(* Logix 5000 project; controller LIgacoesEletricas vendor 1 type 14 code 43 rev 13.1; software revision 13.00 *)

TASK MainTask (continuous, watchdog 500 ms) : MainProgram

MODULES
   Controller : vendor 1 type 14 code 43 (CompactLogixController 0, rev 13.1)
      Local : CompactBus (CompactVirtualAdapter 3, rev 13.1, Input RPI 2 ms)
         M1 : 1769-IQ16 (Compact 1, rev 1.1, Input RPI 2 ms)   // Módulo 1
         M3 : 1769-IQ16 (Compact 3, rev 1.1, Input RPI 2 ms)   // Módulo 3
         M2 : 1769-IQ16 (Compact 2, rev 1.1, Input RPI 2 ms)   // Módulo 2
         M4 : vendor 1 type 7 code 86 (Compact 4, rev 2.1, Output RPI 2 ms)   // Módulo 4
         M5 : vendor 1 type 7 code 86 (Compact 5, rev 2.1, Output RPI 2 ms)   // Módulo 5
         M7 : vendor 1 type 7 code 86 (Compact 7, rev 2.1, Output RPI 2 ms)   // Módulo 7
         M6 : vendor 1 type 7 code 86 (Compact 6, rev 2.1, Output RPI 2 ms)   // Módulo 6
END_MODULES

VAR_GLOBAL   (* controller tags *)
   E0 : ALIAS FOR Local:1:I.Data.0;   // E0 - Entrada do painel
   E1 : ALIAS FOR Local:1:I.Data.1;   // E1 - Entrada do painel
   E1B1 : ALIAS FOR Local:1:I.Data.8;   // E1B1 - indicação de cilindro S1Y1 recuado - alimentação de peças
   E1B2 : ALIAS FOR Local:1:I.Data.9;   // E1B2 - Iindicação do cilindro S1Y1 avançado - alimentação de peças
   E1S1 : ALIAS FOR Local:1:I.Data.10;   // E1S1 - indicação de presença de peças na alimentação
   E1S2 : ALIAS FOR Local:1:I.Data.11;   // E1S2 - indicação de presença de peças fixada na ventosa - oscilador
   E1S3 : ALIAS FOR Local:1:I.Data.12;   // E1S3 - indicação do oscilador (S1Y5) no lado do alimentador
   E1S4 : ALIAS FOR Local:1:I.Data.13;   // E1S4 - indicação do oscilador (S1Y4) no lado do elevador
   E2 : ALIAS FOR Local:1:I.Data.2;   // E2 - Entrada do painel
   E2B1 : ALIAS FOR Local:1:I.Data.14;   // E2B1 - indicação da plataforma (S2Y1) no nível inferior
   E2B2 : ALIAS FOR Local:1:I.Data.15;   // E2B2 - indicação da plataforma (S2Y2) no nível superior
   E2B3 : ALIAS FOR Local:2:I.Data.4;   // E2B3 - indicação do cilindro S2Y3 recuado - descarga de peças na seleção
   E2B4 : ALIAS FOR Local:2:I.Data.5;   // E2B4 - indicação do cilindro S2Y3 avançado - descarga de peças na seleção
   E2B5 : ALIAS FOR Local:2:I.Data.6;   // E2B5 - indicação de peças da cor laranja - sensor ótico - seleção
   E2B6 : ALIAS FOR Local:2:I.Data.7;   // E2B6 - indicação de presença de peças - sensor capacitivo - seleção
   E2B7 : ALIAS FOR Local:2:I.Data.8;   // E2B7 - indicação de peças metálicas - sensor indutivo - seleção
   E3 : ALIAS FOR Local:1:I.Data.3;   // E3 - Entrada do painel
   E3B1 : ALIAS FOR Local:2:I.Data.9;   // E3B1 - indicação de furadeira (S3Y1) na posição superior
   E3B2 : ALIAS FOR Local:2:I.Data.10;   // E3B2 - Iindicação da furadeira (S3Y2) na posição inferior
   E3B3 : ALIAS FOR Local:2:I.Data.0;   // E3B3 - indicação do cilindro S3Y3 recuado - controle de qualidade
   E3B4 : ALIAS FOR Local:2:I.Data.1;   // E3B4 - indicação do cilindro S3Y3 avançado - controle de qualidade
   E3B5 : ALIAS FOR Local:2:I.Data.13;   // E3B5 - indicação do cilindro S3Y4 recuado - fixação de peças na furadeira
   E3B6 : ALIAS FOR Local:2:I.Data.12;   // E3B6 - indicação do cilindro S3Y4 avançado - fixação de peças na furadeira
   E3B7 : ALIAS FOR Local:2:I.Data.11;   // E3B7 - indicação de posicionamento da mesa indexada - sensor indutivo
   E3B8 : ALIAS FOR Local:3:I.Data.3;   // E3B8 - indicação de presença de peças na mesa indexada - descarga da correia transportadora - sensor ótico
   E4 : ALIAS FOR Local:1:I.Data.4;   // E4 - Entrada do painel
   E4B1 : ALIAS FOR Local:2:I.Data.2;   // E4B1 - indicação do cilindro S4Y2 na posição superior - cilindro de transporte de peças para o armazenamento
   E4B2 : ALIAS FOR Local:2:I.Data.3;   // E4B2 - indicação do cilindro S4Y2 na posição inferior - cilindro de transporte de peças para o armazenamento
   E4S2 : ALIAS FOR Local:2:I.Data.14;   // E4S2 - indicação de peças fixada na ventasa - cilindro do armazenamento
   E5 : ALIAS FOR Local:1:I.Data.5;   // E5 - Entrada do painel
   E5B1 : ALIAS FOR Local:3:I.Data.6;   // E5B1 - indicação da ponte transportadora transversal na posição de carregamento (lado S33)
   E5B2 : ALIAS FOR Local:3:I.Data.4;   // E5B2 - indicação da ponte transportadora transversal na posição de descarregamento (lado S32)
   E5B3 : ALIAS FOR Local:3:I.Data.2;   // E5B3 - indicação da ponte transportadora transversal na posição de descarregamento (lado S30)
   E5B4 : ALIAS FOR Local:3:I.Data.1;   // E5B4 - indicação da ponte transportadora longitudinal na posição de descarregamento (lado S30)
   E5B5 : ALIAS FOR Local:3:I.Data.0;   // E5B5 - indicação da ponte transportadora longitudinal na posição de carregamento (lado S31)
   E5B6 : ALIAS FOR Local:3:I.Data.5;   // E5B6 - indicação da ponte transportadora transversal na posição de descarregamento (lado S30)
   E6 : ALIAS FOR Local:1:I.Data.6;   // E6 - Entrada do painel
   E7 : ALIAS FOR Local:1:I.Data.7;   // E7 - Entrada do painel
   S0 : ALIAS FOR Local:4:O.Data.0;   // Saída auxiliar
   S1 : ALIAS FOR Local:4:O.Data.1;   // Saída auxiliar
   S1Y1 : ALIAS FOR Local:5:O.Data.0;   // S1Y1 - cilindro de alimentação de peças
   S1Y2 : ALIAS FOR Local:5:O.Data.1;   // S1Y2 - válvula da ventosa - fixação de peças no oscilador
   S1Y3 : ALIAS FOR Local:5:O.Data.2;   // S1Y3 - válvula da ventosa - liberação de peças do oscilador
   S1Y4 : ALIAS FOR Local:5:O.Data.3;   // S1Y4 - válvula do oscilador - deslocamento para o lado do elevador
   S1Y5 : ALIAS FOR Local:5:O.Data.4;   // S1Y5 - válvula do oscilador - deslocamento para o lado da alimentação
   S2 : ALIAS FOR Local:4:O.Data.2;   // Saída auxiliar
   S2Y1 : ALIAS FOR Local:5:O.Data.5;   // S2Y1 - válvula do elevador - deslocamento da para o nível inferior
   S2Y2 : ALIAS FOR Local:5:O.Data.6;   // S2Y2 - válvula do elevador - deslocamento da para o nível superior
   S2Y3 : ALIAS FOR Local:5:O.Data.7;   // S2Y3 - válvula da descarga na seleção de peças
   S3 : ALIAS FOR Local:4:O.Data.3;   // Saída auxiliar
   S3Y1 : ALIAS FOR Local:6:O.Data.6;   // S3Y1 - válvula da furadeira - movimento para posição inferior
   S3Y2 : ALIAS FOR Local:6:O.Data.7;   // S3Y2 - válvula da furadeira - movimento para posição superior
   S3Y3 : ALIAS FOR Local:6:O.Data.5;   // S3Y3 - válvula do controle de qualidade
   S3Y4 : ALIAS FOR Local:6:O.Data.4;   // S3Y4 - válvula do cilindro de fixação de peças para furação
   S4 : ALIAS FOR Local:4:O.Data.4;   // Saída auxiliar
   S4Y1 : ALIAS FOR Local:6:O.Data.2;   // S4Y1 - válvula do cilindro de transporte de peças para o armazenamento - movimento para posição inferior
   S4Y2 : ALIAS FOR Local:6:O.Data.3;   // S4Y2 - válvula do cilindro de transporte de peças para o armazenamento - movimento para posição superior
   S4Y3 : ALIAS FOR Local:6:O.Data.1;   // S4Y3 - válvula da ventosa do transporte de peças para o armazenamento - fixação de peça
   S4Y4 : ALIAS FOR Local:6:O.Data.0;   // S4Y4 - válvula da ventosa do transporte de peças para o armazenamento - liberação da peça
   S5 : ALIAS FOR Local:4:O.Data.5;   // Saída auxiliar
   S6 : ALIAS FOR Local:4:O.Data.6;   // Saída auxiliar
   S7 : ALIAS FOR Local:4:O.Data.7;   // Saída auxiliar
   SK1M1 : ALIAS FOR Local:7:O.Data.6;   // SK1M1 - relé do motor da furadeira
   SK2M2 : ALIAS FOR Local:7:O.Data.5;   // SK2M2 - relé do motor da mesa indexada
   SK3M3 : ALIAS FOR Local:7:O.Data.4;   // SK3M3 - relé do motor da correia transportadora
   SK4M4 : ALIAS FOR Local:7:O.Data.2;   // SK4M4 - relé do motor do movimento transversal da ponte transportadora para S33
   SK5M4 : ALIAS FOR Local:7:O.Data.3;   // SK5M4 - relé do motor do movimento transversal da ponte transportadora para S32
   SK6M5 : ALIAS FOR Local:7:O.Data.0;   // SK6M5 - relé do motor do movimento longitudinal da ponte transportadora para S31
   SK7M5 : ALIAS FOR Local:7:O.Data.1;   // SK7M5 - relé do motor do movimento longitudinal da ponte transportadora para S30
END_VAR

PROGRAM MainProgram   (* routine attr 65 MainRoutine *)
VAR
   armazena : BOOL;
   aux1 : BOOL;
   aux2 : BOOL;
   fim_do_teste : BOOL;
   inicia_depuracao : BOOL := 1;
   Passo1 : BOOL;
   Passo10 : BOOL;
   Passo11 : BOOL;
   Passo12 : BOOL;
   Passo13 : BOOL;
   Passo14 : BOOL;
   Passo15 : BOOL;
   Passo16 : BOOL;
   Passo17 : BOOL;
   Passo18 : BOOL;
   Passo19 : BOOL;
   Passo2 : BOOL;
   Passo20 : BOOL;
   Passo21 : BOOL;
   Passo22 : BOOL;
   Passo23 : BOOL;
   Passo24 : BOOL;
   Passo25 : BOOL;
   Passo26 : BOOL;
   Passo27 : BOOL;
   Passo28 : BOOL;
   Passo29 : BOOL;
   Passo3 : BOOL;
   Passo30 : BOOL;
   Passo31 : BOOL;
   Passo32 : BOOL;
   Passo33 : BOOL;
   Passo34 : BOOL;
   Passo35 : BOOL;
   Passo36 : BOOL;
   Passo37 : BOOL;
   Passo38 : BOOL;
   Passo39 : BOOL;
   Passo4 : BOOL;
   Passo5 : BOOL;
   Passo6 : BOOL;
   Passo7 : BOOL;
   Passo8 : BOOL;
   Passo9 : BOOL;
   peca_laranja : BOOL;
   peca_metalica : BOOL;
   saidaosr : BOOL;
   tempo : TIMER := (PRE := 2000);
   temporizador1 : TIMER := (PRE := 6000);
END_VAR

ROUTINE MainRoutine   (* ladder *)
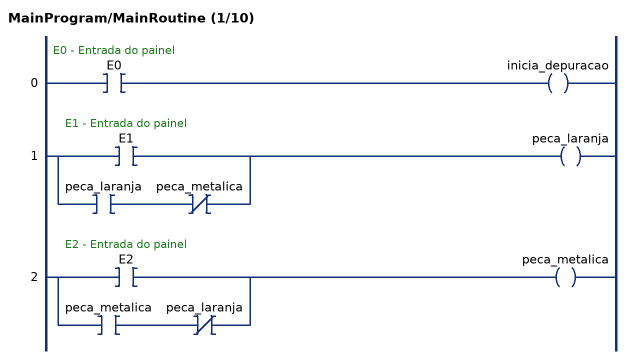
   0: XIC(E0)OTE(inicia_depuracao);
   1: [XIC(E1) ,XIC(peca_laranja) XIO(peca_metalica) ]OTE(peca_laranja);
   2: [XIC(E2) ,XIC(peca_metalica) XIO(peca_laranja) ]OTE(peca_metalica);
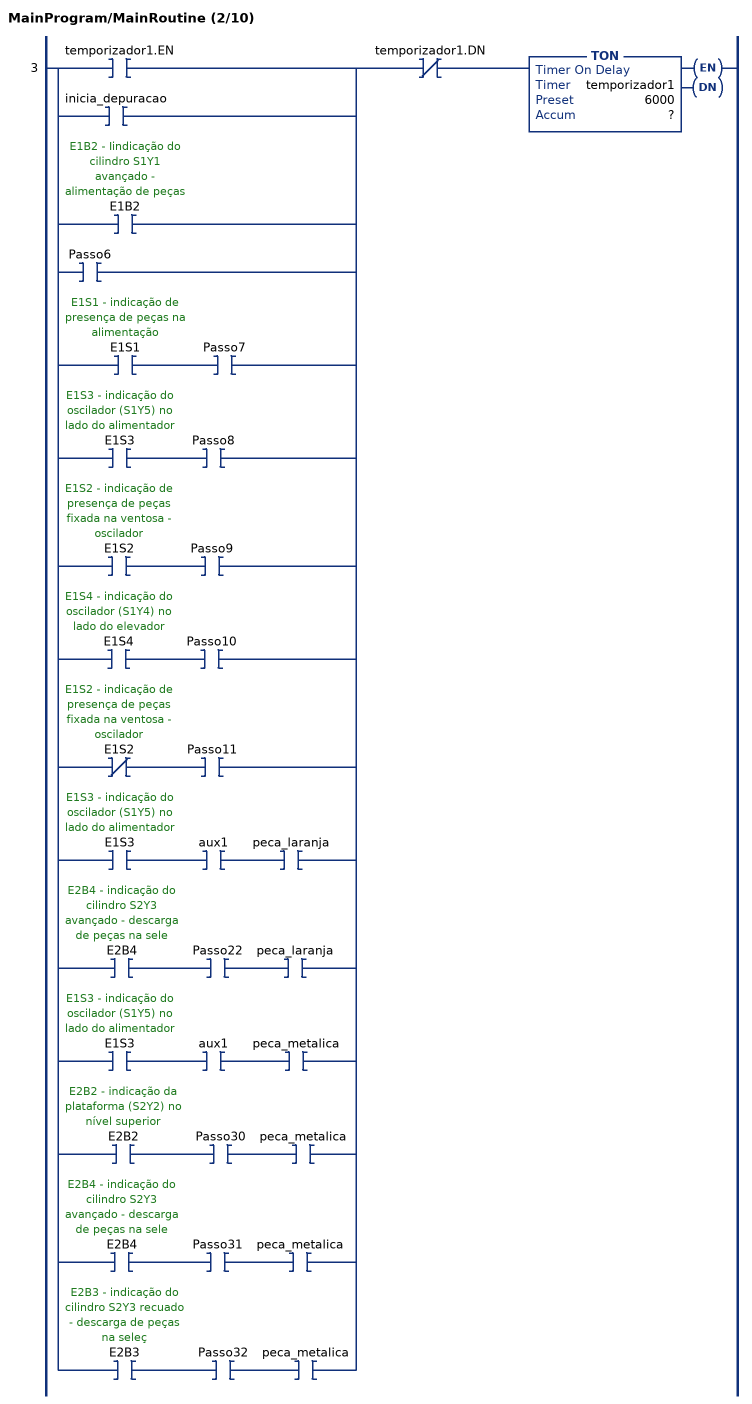
   3: [XIC(temporizador1.EN) ,XIC(inicia_depuracao) ,XIC(E1B2) ,XIC(Passo6) ,XIC(E1S1) XIC(Passo7) ,XIC(E1S3) XIC(Passo8) ,XIC(E1S2) XIC(Passo9) ,XIC(E1S4) XIC(Passo10) ,XIO(E1S2) XIC(Passo11) ,XIC(E1S3) XIC(aux1) XIC(peca_laranja) ,XIC(E2B4) XIC(Passo22) XIC(peca_laranja) ,XIC(E1S3) XIC(aux1) XIC(peca_metalica) ,XIC(E2B2) XIC(Passo30) XIC(peca_metalica) ,XIC(E2B4) XIC(Passo31) XIC(peca_metalica) ,XIC(E2B3) XIC(Passo32) XIC(peca_metalica) ]XIO(temporizador1.DN)TON(temporizador1,?,?);
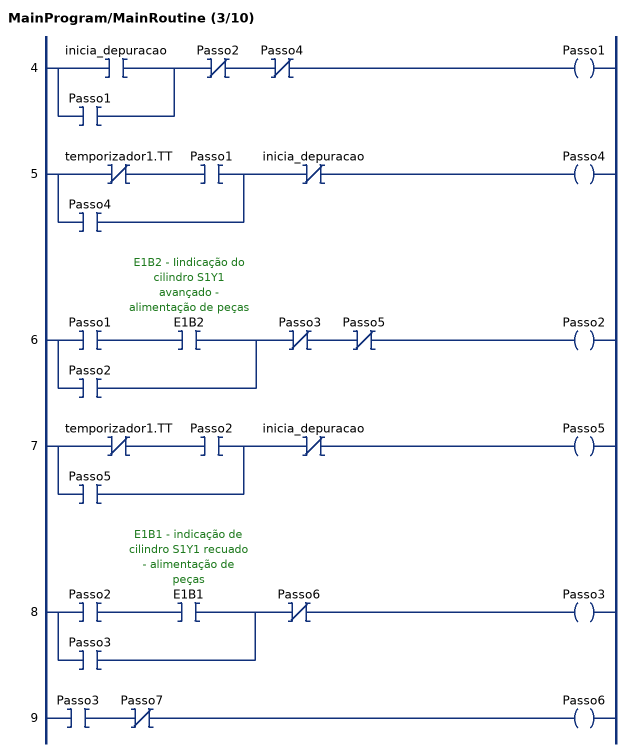
   4: [XIC(inicia_depuracao) ,XIC(Passo1) ]XIO(Passo2)XIO(Passo4)OTE(Passo1);
   5: [XIO(temporizador1.TT) XIC(Passo1) ,XIC(Passo4) ]XIO(inicia_depuracao)OTE(Passo4);
   6: [XIC(Passo1) XIC(E1B2) ,XIC(Passo2) ]XIO(Passo3)XIO(Passo5)OTE(Passo2);
   7: [XIO(temporizador1.TT) XIC(Passo2) ,XIC(Passo5) ]XIO(inicia_depuracao)OTE(Passo5);
   8: [XIC(Passo2) XIC(E1B1) ,XIC(Passo3) ]XIO(Passo6)OTE(Passo3);
   9: XIC(Passo3)XIO(Passo7)OTE(Passo6);
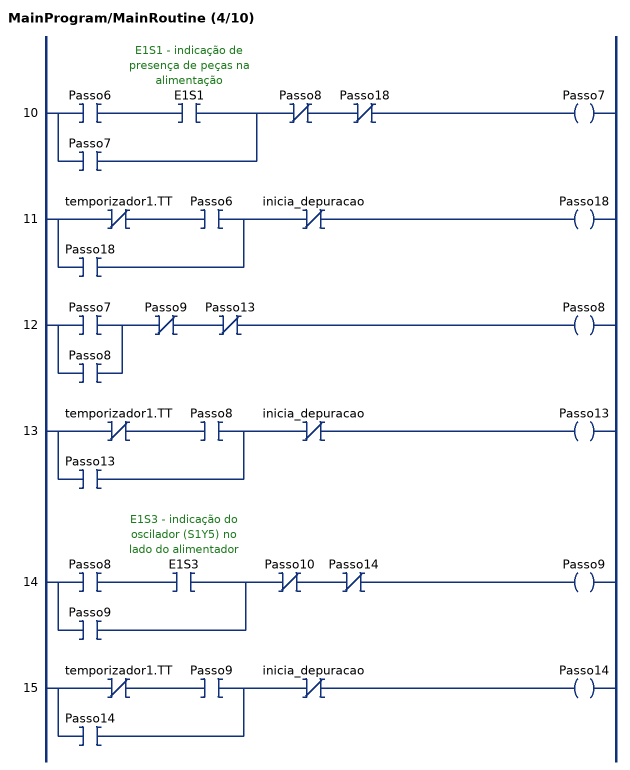
   10: [XIC(Passo6) XIC(E1S1) ,XIC(Passo7) ]XIO(Passo8)XIO(Passo18)OTE(Passo7);
   11: [XIO(temporizador1.TT) XIC(Passo6) ,XIC(Passo18) ]XIO(inicia_depuracao)OTE(Passo18);
   12: [XIC(Passo7) ,XIC(Passo8) ]XIO(Passo9)XIO(Passo13)OTE(Passo8);
   13: [XIO(temporizador1.TT) XIC(Passo8) ,XIC(Passo13) ]XIO(inicia_depuracao)OTE(Passo13);
   14: [XIC(Passo8) XIC(E1S3) ,XIC(Passo9) ]XIO(Passo10)XIO(Passo14)OTE(Passo9);
   15: [XIO(temporizador1.TT) XIC(Passo9) ,XIC(Passo14) ]XIO(inicia_depuracao)OTE(Passo14);
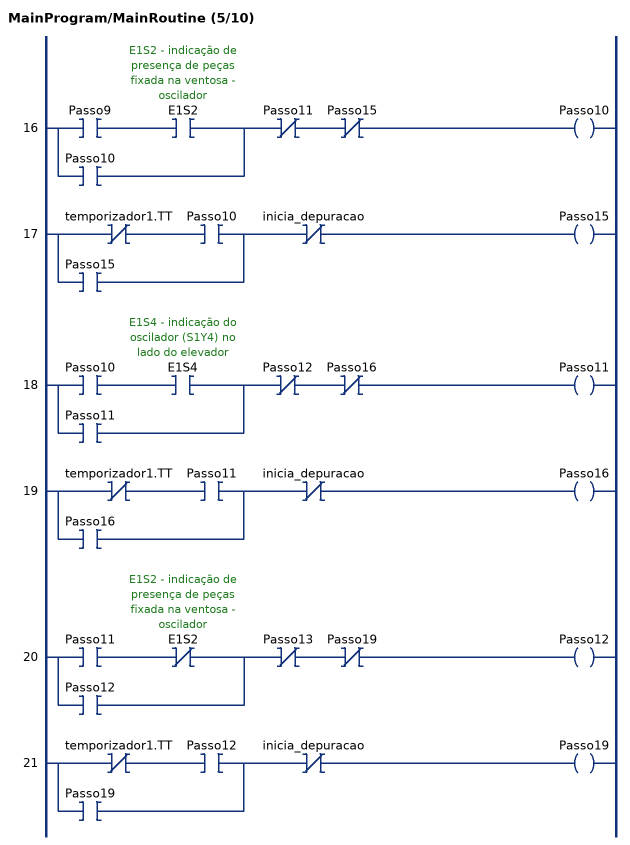
   16: [XIC(Passo9) XIC(E1S2) ,XIC(Passo10) ]XIO(Passo11)XIO(Passo15)OTE(Passo10);
   17: [XIO(temporizador1.TT) XIC(Passo10) ,XIC(Passo15) ]XIO(inicia_depuracao)OTE(Passo15);
   18: [XIC(Passo10) XIC(E1S4) ,XIC(Passo11) ]XIO(Passo12)XIO(Passo16)OTE(Passo11);
   19: [XIO(temporizador1.TT) XIC(Passo11) ,XIC(Passo16) ]XIO(inicia_depuracao)OTE(Passo16);
   20: [XIC(Passo11) XIO(E1S2) ,XIC(Passo12) ]XIO(Passo13)XIO(Passo19)OTE(Passo12);
   21: [XIO(temporizador1.TT) XIC(Passo12) ,XIC(Passo19) ]XIO(inicia_depuracao)OTE(Passo19);
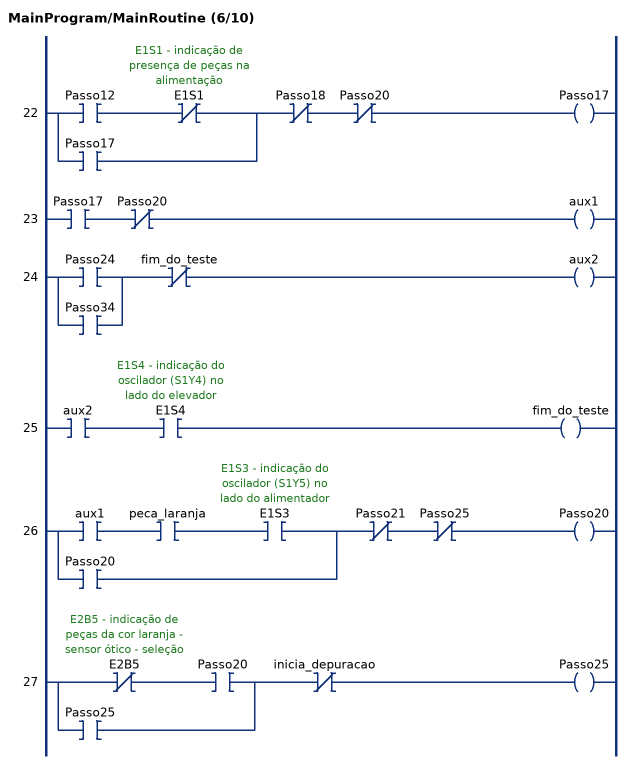
   22: [XIC(Passo12) XIO(E1S1) ,XIC(Passo17) ]XIO(Passo18)XIO(Passo20)OTE(Passo17);
   23: XIC(Passo17)XIO(Passo20)OTE(aux1);
   24: [XIC(Passo24) ,XIC(Passo34) ]XIO(fim_do_teste)OTE(aux2);
   25: XIC(aux2)XIC(E1S4)OTE(fim_do_teste);
   26: [XIC(aux1) XIC(peca_laranja) XIC(E1S3) ,XIC(Passo20) ]XIO(Passo21)XIO(Passo25)OTE(Passo20);
   27: [XIO(E2B5) XIC(Passo20) ,XIC(Passo25) ]XIO(inicia_depuracao)OTE(Passo25);
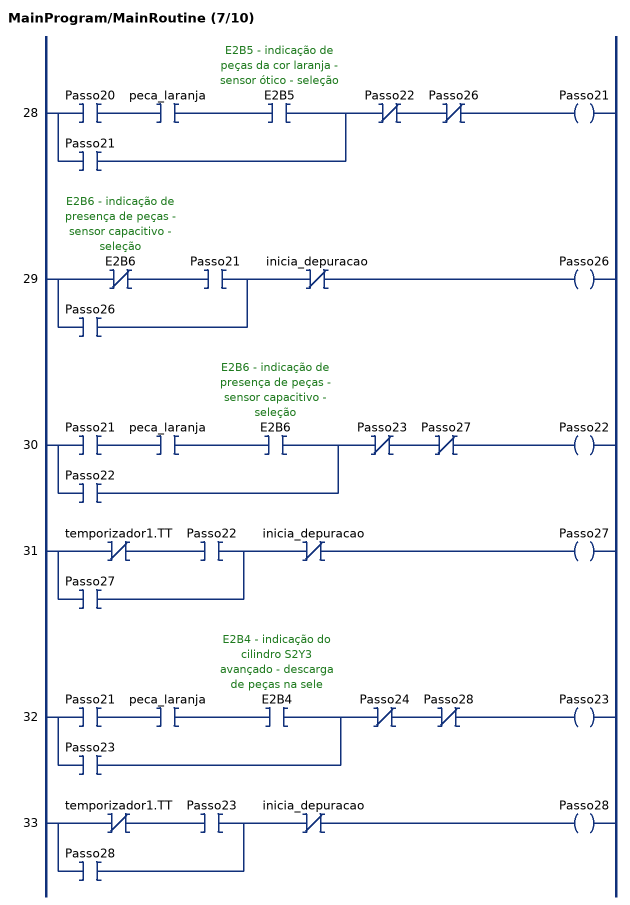
   28: [XIC(Passo20) XIC(peca_laranja) XIC(E2B5) ,XIC(Passo21) ]XIO(Passo22)XIO(Passo26)OTE(Passo21);
   29: [XIO(E2B6) XIC(Passo21) ,XIC(Passo26) ]XIO(inicia_depuracao)OTE(Passo26);
   30: [XIC(Passo21) XIC(peca_laranja) XIC(E2B6) ,XIC(Passo22) ]XIO(Passo23)XIO(Passo27)OTE(Passo22);
   31: [XIO(temporizador1.TT) XIC(Passo22) ,XIC(Passo27) ]XIO(inicia_depuracao)OTE(Passo27);
   32: [XIC(Passo21) XIC(peca_laranja) XIC(E2B4) ,XIC(Passo23) ]XIO(Passo24)XIO(Passo28)OTE(Passo23);
   33: [XIO(temporizador1.TT) XIC(Passo23) ,XIC(Passo28) ]XIO(inicia_depuracao)OTE(Passo28);
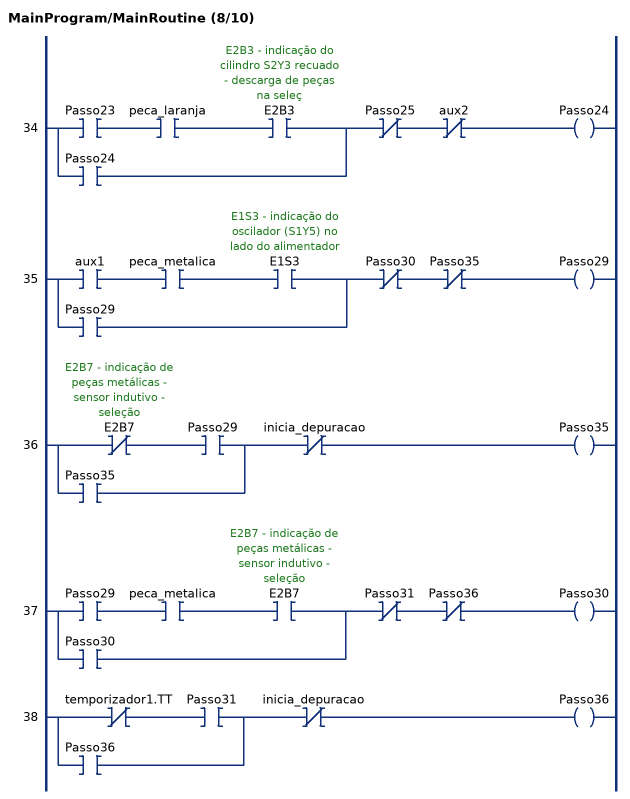
   34: [XIC(Passo23) XIC(peca_laranja) XIC(E2B3) ,XIC(Passo24) ]XIO(Passo25)XIO(aux2)OTE(Passo24);
   35: [XIC(aux1) XIC(peca_metalica) XIC(E1S3) ,XIC(Passo29) ]XIO(Passo30)XIO(Passo35)OTE(Passo29);
   36: [XIO(E2B7) XIC(Passo29) ,XIC(Passo35) ]XIO(inicia_depuracao)OTE(Passo35);
   37: [XIC(Passo29) XIC(peca_metalica) XIC(E2B7) ,XIC(Passo30) ]XIO(Passo31)XIO(Passo36)OTE(Passo30);
   38: [XIO(temporizador1.TT) XIC(Passo31) ,XIC(Passo36) ]XIO(inicia_depuracao)OTE(Passo36);
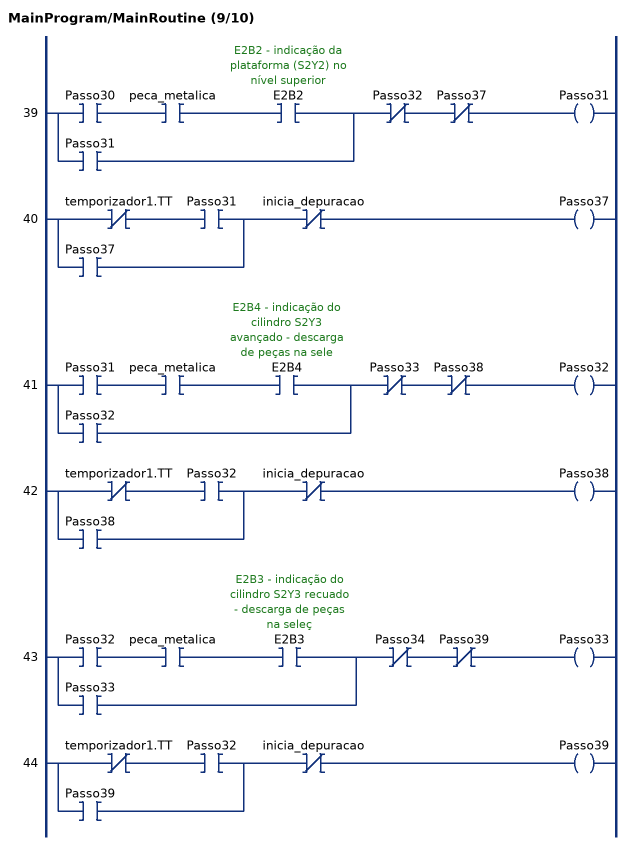
   39: [XIC(Passo30) XIC(peca_metalica) XIC(E2B2) ,XIC(Passo31) ]XIO(Passo32)XIO(Passo37)OTE(Passo31);
   40: [XIO(temporizador1.TT) XIC(Passo31) ,XIC(Passo37) ]XIO(inicia_depuracao)OTE(Passo37);
   41: [XIC(Passo31) XIC(peca_metalica) XIC(E2B4) ,XIC(Passo32) ]XIO(Passo33)XIO(Passo38)OTE(Passo32);
   42: [XIO(temporizador1.TT) XIC(Passo32) ,XIC(Passo38) ]XIO(inicia_depuracao)OTE(Passo38);
   43: [XIC(Passo32) XIC(peca_metalica) XIC(E2B3) ,XIC(Passo33) ]XIO(Passo34)XIO(Passo39)OTE(Passo33);
   44: [XIO(temporizador1.TT) XIC(Passo32) ,XIC(Passo39) ]XIO(inicia_depuracao)OTE(Passo39);
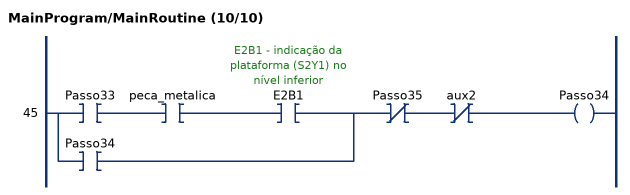
   45: [XIC(Passo33) XIC(peca_metalica) XIC(E2B1) ,XIC(Passo34) ]XIO(Passo35)XIO(aux2)OTE(Passo34);
END_ROUTINE
END_PROGRAM
